{attribute 'GeneratedUsingTerminal: EL1502-0000-0018'}
{attribute addProperty BoxType "EL1502-0000-0018"}
{attribute addProperty Id "ControlAT %Q*Control_854091F64Set_counter_valueAT %Q*UDINT4"}
{attribute addProperty CRC "1166031278"}
{attribute addProperty Size "8"}
TYPE CNT_Outputs_458039AE :
STRUCT
	{attribute addProperty Name "Control"}
	Control AT %Q* : Control_854091F6;
	{attribute addProperty Name "Set_counter_value"}
	Set_counter_value AT %Q* : UDINT;
END_STRUCT
END_TYPE

(* stored: Version 1.2.0.0, ProductVersion 3.1.4024.9
   DUT CNT_Outputs_458039AE: Id {f151e0dd-4dd8-4cd4-81bf-378fbc4d218f} *)
